(* IEC 61131-3 sources: FibonacciChallenge/Class/MyFirstClass, 1 file *)

(* ---- MyFirstClass.st ---- *)
(*!
<Class
	Name               = "MyFirstClass"
	Revision           = "0.0"
	RealtimeTask       = "false"
	CyclicTask         = "true"
	BackgroundTask     = "false"
	Sigmatek           = "false"
	OSInterface        = "false"
	HighPriority       = "false"
	Automatic          = "false"
	UpdateMode         = "Prescan"
	SharedCommandTable = "true"
	Objectsize         = "(284,120)">
	<Channels>
		<Server Name="ClassSvr" Visualized="false" Initialize="false" WriteProtected="true" Retentive="false"/>
		<Server Name="Speed" Visualized="false" Initialize="false" WriteProtected="false" Retentive="false"/>
		<Client Name="o_Led1" Required="true" Internal="false"/>
		<Client Name="o_Led2" Required="true" Internal="false"/>
		<Client Name="o_Led3" Required="true" Internal="false"/>
		<Client Name="o_Led4" Required="true" Internal="false"/>
	</Channels>
</Class>
*)
MyFirstClass : CLASS
  //Servers:
	ClassSvr 	: SvrChCmd_DINT;
	Speed 	: SvrCh_UDINT;
  //Clients:
	o_Led1 	: CltCh_DINT;
	o_Led2 	: CltCh_DINT;
	o_Led3 	: CltCh_DINT;
	o_Led4 	: CltCh_DINT;
  //Variables:
		Stepper 	: DINT;
		udTimeMark 	: UDINT;
		Value 	: BOOL;
  //Functions:

	FUNCTION VIRTUAL GLOBAL Init;

	FUNCTION VIRTUAL GLOBAL CyWork
		VAR_INPUT
			EAX 	: UDINT;
		END_VAR
		VAR_OUTPUT
			state (EAX) 	: UDINT;
		END_VAR;
  //Tables:
	FUNCTION @STD
		VAR_OUTPUT
			ret_code	: CONFSTATES;
		END_VAR;
	FUNCTION GLOBAL TAB @CT_;
END_CLASS;

FUNCTION VIRTUAL GLOBAL MyFirstClass::Init

Speed := 1000;
Value := 1;

END_FUNCTION

FUNCTION VIRTUAL GLOBAL MyFirstClass::CyWork
	VAR_INPUT
		EAX 	: UDINT;
	END_VAR
	VAR_OUTPUT
		state (EAX) 	: UDINT;
	END_VAR

  if ops.tAbsolute > (udTimeMark + Speed) then

    Value := !!Value;
    o_Led1.Write(Value);
    udTimeMark := ops.tAbsolute;
  end_if;

	state := READY;

END_FUNCTION
